Fanuc KAREL source: ko00052.KL

PROGRAM KO00052
%STACKSIZE=65535
%PRIORITY=65535
%NOLOCKGROUP
VAR
P1 : XYZWPR
P2 : POSITION
F : BOOLEAN
OUT : JOINTPOS9
BEGIN
F=TRUE
-- UNSAFE_SOURCE_IR line 11: CALL_RESULT MIRROR(convert_xyzwpr_to_xyzwprext(P1), P2, F)
END KO00052
